INTERFACE Motor

METHOD SetSpeed : BOOL
VAR_INPUT
	 newFreq : REAL;
END_VAR
END_METHOD

END_INTERFACE

(* stored: Version 1.1.0.1, ProductVersion 3.1.4024.16
   Itf Motor: Id {4d96e211-9f67-4647-98db-b86a39601f8d}
   Method SetSpeed: Id {2c8dec59-44e2-4517-9e1f-08e61ec38aa0} *)
